{attribute 'GeneratedUsingTerminal: EK1122-0000-0018'}
{attribute addProperty BoxType "EK1122-0000-0018"}
{attribute addProperty Id "Beckhoff_EK12xxsub_EK1100EK1100_AB5A94672"}
{attribute addProperty CRC "503763487"}
{attribute addProperty Size "2"}
TYPE Beckhoff_EK12xxEK1122_1E06D21F EXTENDS EK1122_AB5A9467 :
STRUCT
	{attribute addProperty Name "Beckhoff_EK12xxsub_EK1100"}
	{attribute addProperty PreviousPort "Beckhoff EK12xxEK1122 : D"}
	Beckhoff_EK12xxsub_EK1100 : EK1100_AB5A9467;
END_STRUCT
END_TYPE

(* stored: Version 1.2.0.0, ProductVersion 3.1.4024.9
   DUT Beckhoff_EK12xxEK1122_1E06D21F: Id {0a09c77b-55ef-487d-8383-dc4cdd23c6f6} *)
